FUNCTION F_DecimalData : LREAL
VAR_INPUT
	
	f_value_input : REAL;
	// decimal places
	n_decimal_digit : INT;
	// Round or not
	b_round_data: BOOL;

END_VAR
VAR_OUTPUT	
	f_value_output : REAL;
END_VAR
VAR
END_VAR

f_value_output := STRING_TO_REAL(LREAL_TO_FMTSTR(TO_REAL(f_value_input), n_decimal_digit, b_round_data));
F_DecimalData := f_value_output

END_FUNCTION

(* stored: Version 1.1.0.1, ProductVersion 3.1.4024.11
   POU F_DecimalData: Id {66d33ad8-e83a-4919-8f59-cd46dd00ddc3}, SpecialFunc None *)
